# EPICS StreamDevice protocol: linkam95Sup/devlinkam95.proto
OutTerminator = CR;
InTerminator  = CR;
#
# From Diamond T92-94 protocol
#
#replytimeout = 1000;
#readtimeout  = 500;
#locktimeout = 5000;
#extrainput   = Ignore;
#separator = "";

getStatus {
	out "T";
	in "%10c";
}

getStatusInitial {
    out "T";
	in "%1r"
	   "%(\$1IN_ERROR)1r"
	   "%(\$1IN_PUMP_STAT)1r"
	   "\?\?\?"
	   "%(\$1IN_TEMP)4r";
}

getStatusBackup {
    out "T";
	in "%1r"
	   "%(\$1IN_ERROR)1r"
	   "%(\$1IN_PUMP_STAT)1r"
	   "(\$1IN_DUMMY)3r"
	   "%(\$1IN_TEMP)4r";
}

setRate {
	out "R1%04u";
}

setLimit {
	out "L1%04i";
}

# Stop(E)/Start(S) Temperature control
setRampControl {
	out "%{E|S}";
}

# Force heating (H), force cooling (C), or hold at current temperature (O)
setForceRamp {
	out "%{H|C|O}";
}

# Select LNP manual (Pm0) or automatic mode (Pa0)
setPumpMode {
	out "%{Pm0|Pa0}";
}

# Select LNP speed (in manual mode only)
setPumpSpeed {
	out "P%{0|1|2|3|4|5|6|7|8|9|:|;|<|=|>|?|@|A|B|C|D|E|F|G|H|I|J|K|L|M|N}";
}
